FUNCTION_BLOCK ComponentCollection_TEST
VAR

END_VAR

CollectionAddsComponentSucessfully();
CollectionRejectsAddingComponentDuplicate();
CollectionRejectsAddingNullComponent();
CollectionRejectsAddingTooManyComponents();
CollectionRejectsRemoveWhenEmpty();
CollectionRejectsRemoveWhenNotFound();
CollectionRejectsRemovingNullComponent();
CollectionReturnsComponentByName();
CollectionRemovesComponentSuccessfully();
CollectionGetItemAtIndex();
CollectionGetCount();

METHOD CollectionAddsComponentSucessfully
VAR
	Expected			: BOOL := TRUE;
	Actual				: BOOL;
	ComponentCollection : ComponentCollection<ApplicationBaseParameter.MaxCountInCollections>;
	Component			: CyclicComponent_Mockup(Name := 'Component 1');
END_VAR
IF TestSuite.Test(__POUNAME()).ExecuteTest() THEN
	Actual := ComponentCollection.AddComponent(Component) = RegistrationResult.Succeeded;
	TestSuite.Test(__POUNAME()).AssertEqual(Expected, Actual);
END_IF
END_METHOD

METHOD CollectionGetCount
VAR
	Expected			: UDINT;
	Actual				: UDINT;
	ComponentCollection : ComponentCollection<ApplicationBaseParameter.MaxCountInCollections>;
	Component			: CyclicComponent_Mockup(Name := 'Component 1');
END_VAR
IF TestSuite.Test(__POUNAME()).ExecuteTest() THEN
	Expected := 1;
	ComponentCollection.AddComponent(Component);
	Actual := ComponentCollection.Count;
	TestSuite.Test(__POUNAME()).AssertEqual(Expected, Actual);
END_IF
END_METHOD

METHOD CollectionGetItemAtIndex
VAR
	Expected			: BOOL := TRUE;
	Actual				: BOOL;
	ComponentCollection : ComponentCollection<2>;
	Component1			: CyclicComponent_Mockup(Name := 'Component 1');
	Component2			: CyclicComponent_Mockup(Name := 'Component 2');
	ReturnedComponent	: I_Component;
END_VAR
IF TestSuite.Test(__POUNAME()).ExecuteTest() THEN
	ComponentCollection.AddComponent(Component1);
	ComponentCollection.AddComponent(Component2);
	ReturnedComponent := ComponentCollection.GetAtIndex(1);
	Actual			  := ReturnedComponent.Name = Component2.Name;
	TestSuite.Test(__POUNAME()).AssertEqual(Expected, Actual);
END_IF
END_METHOD

METHOD CollectionRejectsAddingComponentDuplicate
VAR
	Expected	   : BOOL := TRUE;
	Actual		   : BOOL;
	ComponentCollection : ComponentCollection<ApplicationBaseParameter.MaxCountInCollections>;
	Component			: CyclicComponent_Mockup(Name := 'Component 1');
END_VAR
IF TestSuite.Test(__POUNAME()).ExecuteTest() THEN
	ComponentCollection.AddComponent(Component);
	Actual := ComponentCollection.AddComponent(Component) = RegistrationResult.AlreadyAdded;
	TestSuite.Test(__POUNAME()).AssertEqual(Expected, Actual);
END_IF
END_METHOD

METHOD CollectionRejectsAddingNullComponent
VAR
	Expected	   : BOOL := TRUE;
	Actual		   : BOOL;
	ComponentCollection : ComponentCollection<ApplicationBaseParameter.MaxCountInCollections>;
END_VAR
IF TestSuite.Test(__POUNAME()).ExecuteTest() THEN
	Actual := ComponentCollection.AddComponent(16#0) = RegistrationResult.NullReference;
	TestSuite.Test(__POUNAME()).AssertEqual(Expected, Actual);
END_IF
END_METHOD

METHOD CollectionRejectsAddingTooManyComponents
VAR
	Expected	   : BOOL := TRUE;
	Actual		   : BOOL;
	ComponentCollection : ComponentCollection<1>;
	Component1			: CyclicComponent_Mockup(Name := 'Component 1');
	Component2			: CyclicComponent_Mockup(Name := 'Component 2');
END_VAR
IF TestSuite.Test(__POUNAME()).ExecuteTest() THEN
	ComponentCollection.AddComponent(Component1);
	Actual := ComponentCollection.AddComponent(Component2) = RegistrationResult.TooManyComponents;
	TestSuite.Test(__POUNAME()).AssertEqual(Expected, Actual);
END_IF
END_METHOD

METHOD CollectionRejectsRemoveWhenEmpty
VAR
	Expected	   : BOOL := TRUE;
	Actual		   : BOOL;
	ComponentCollection : ComponentCollection<ApplicationBaseParameter.MaxCountInCollections>;
	Component			: CyclicComponent_Mockup(Name := 'Component 1');
END_VAR
IF TestSuite.Test(__POUNAME()).ExecuteTest() THEN
	Actual := ComponentCollection.RemoveComponent(Component) = RegistrationResult.CollectionEmpty;
	TestSuite.Test(__POUNAME()).AssertEqual(Expected, Actual);
END_IF
END_METHOD

METHOD CollectionRejectsRemoveWhenNotFound
VAR
	Expected	   : BOOL := TRUE;
	Actual		   : BOOL;
	ComponentCollection : ComponentCollection<1>;
	Component1			: CyclicComponent_Mockup(Name := 'Component 1');
	Component2			: CyclicComponent_Mockup(Name := 'Component 2');
END_VAR
IF TestSuite.Test(__POUNAME()).ExecuteTest() THEN
	ComponentCollection.AddComponent(Component1);
	Actual := ComponentCollection.RemoveComponent(Component2) = RegistrationResult.NotFoundInCollection;
	TestSuite.Test(__POUNAME()).AssertEqual(Expected, Actual);
END_IF
END_METHOD

METHOD CollectionRejectsRemovingNullComponent
VAR
	Expected	   : BOOL := TRUE;
	Actual		   : BOOL;
	ComponentCollection : ComponentCollection<ApplicationBaseParameter.MaxCountInCollections>;
END_VAR
IF TestSuite.Test(__POUNAME()).ExecuteTest() THEN
	Actual := ComponentCollection.RemoveComponent(16#0) = RegistrationResult.NullReference;
	TestSuite.Test(__POUNAME()).AssertEqual(Expected, Actual);
END_IF
END_METHOD

METHOD CollectionRemovesComponentSuccessfully
VAR
	Expected			: BOOL := TRUE;
	Actual				: BOOL;
	ComponentCollection : ComponentCollection<ApplicationBaseParameter.MaxCountInCollections>;
	Component			: CyclicComponent_Mockup(Name := 'Component 1');
	AddedComponent		: I_Component := Component;
	CollectionComponent : I_Component;
END_VAR
IF TestSuite.Test(__POUNAME()).ExecuteTest() THEN
	ComponentCollection.AddComponent(Component);
	CollectionComponent := ComponentCollection.GetComponentByName('Component 1');
	IF CollectionComponent = AddedComponent THEN
		Actual := ComponentCollection.RemoveComponent(Component) = RegistrationResult.Succeeded;
	END_IF
	TestSuite.Test(__POUNAME()).AssertEqual(Expected, Actual);
END_IF
END_METHOD

METHOD CollectionReturnsComponentByName
VAR
	Expected	   : STRING := 'Component 1';
	Actual		   : STRING;
	ComponentCollection : ComponentCollection<ApplicationBaseParameter.MaxCountInCollections>;
	Component			: CyclicComponent_Mockup(Name := 'Component 1');
END_VAR
IF TestSuite.Test(__POUNAME()).ExecuteTest() THEN
	ComponentCollection.AddComponent(Component);
	Actual := ComponentCollection.GetComponentByName(Expected).Name;
	TestSuite.Test(__POUNAME()).AssertEqual(Expected, Actual);
END_IF
END_METHOD

END_FUNCTION_BLOCK

(* stored: Version 1.1.0.1, ProductVersion 3.1.4026.18
   POU ComponentCollection_TEST: Id {e3340b3a-1f47-411e-8cf3-592998e732d3}, SpecialFunc None
   Method CollectionAddsComponentSucessfully: Id {7ec61a68-feef-4afa-9c67-66271e8ef843}
   Method CollectionGetCount: Id {5b1ce18c-d96c-4f15-8dee-2e504a5dd2c3}
   Method CollectionGetItemAtIndex: Id {6a520ef9-32d2-4c4e-97b0-72b71a124044}
   Method CollectionRejectsAddingComponentDuplicate: Id {ab12516f-81ad-44f7-9c61-e577d843f2f6}
   Method CollectionRejectsAddingNullComponent: Id {4bf860c3-8cd5-43d8-92d8-ab0de04135f2}
   Method CollectionRejectsAddingTooManyComponents: Id {e3170356-2bf3-4f6a-bb76-f0fb8c845f0a}
   Method CollectionRejectsRemoveWhenEmpty: Id {a105872f-e488-4478-9074-219be1266bb2}
   Method CollectionRejectsRemoveWhenNotFound: Id {f5b296ac-e254-4762-ba66-073dcecd396f}
   Method CollectionRejectsRemovingNullComponent: Id {bb5487a6-9114-4666-bb94-b52d1246decc}
   Method CollectionRemovesComponentSuccessfully: Id {a7c852a9-afa2-4cc8-9983-0b8abec4032e}
   Method CollectionReturnsComponentByName: Id {2b07c489-b6c2-4148-83b1-220f4c152bb1} *)
